{attribute 'GeneratedUsingTerminal: IODEVICETYPE_ETHERCATPROT'}
{attribute addProperty BoxType "IODEVICETYPE_ETHERCATPROT"}
{attribute addProperty Id "Beckhoff_APS1xxxBeckhoff_APS1xxx_D211951F586Beckhoff_APS4xxxBeckhoff_APS4xxx_28EA972F604SyncUnitsSyncUnits_99E584AF18InputsInputs_25A0042B160OutputsOutputs_2397A10E106InfoDataInfoData_E68C61CD28"}
{attribute addProperty CRC "3229625005"}
{attribute addProperty Size "1502"}
TYPE EtherCAT_Master_APSxxxx_C0802AAD :
STRUCT
	{attribute addProperty Name "Beckhoff_APS1xxx"}
	{attribute addProperty PreviousPort "EtherCAT_Master_APSxxxx : Master"}
	Beckhoff_APS1xxx : Beckhoff_APS1xxx_D211951F;
	{attribute addProperty Name "Beckhoff_APS4xxx"}
	{attribute addProperty PreviousPort "Beckhoff APS1xxx : C"}
	Beckhoff_APS4xxx : Beckhoff_APS4xxx_28EA972F;
	{attribute addProperty Name "SyncUnits"}
	SyncUnits : SyncUnits_99E584AF;
	{attribute addProperty Name "Inputs"}
	Inputs : Inputs_25A0042B;
	{attribute addProperty Name "Outputs"}
	Outputs : Outputs_2397A10E;
	{attribute addProperty Name "InfoData"}
	InfoData : InfoData_E68C61CD;
END_STRUCT
END_TYPE

(* stored: Version 1.2.0.0, ProductVersion 3.1.4024.9
   DUT EtherCAT_Master_APSxxxx_C0802AAD: Id {15886f89-bfeb-4f91-a951-e4ef190c2499} *)
